Staubli VAL3: BackHomePage.pgx

public program BackHomePage(joint x_jHome, tool x_tTool, mdesc x_mHome)
  local num l_nKey
  local string l_sButton[2]
  local num l_i
  local bool l_bHomeDone
  local bool l_bExit
  local string l_sYesNo
begin
  //-----------------------------------------------------------------------
  //Header begin
  //Description of program
  //  手臂回零页面
  //  F1:终止回零
  //Input parameters
  //
  //Output paramaters
  //Example
  //  call BackHomePage()
  //History
  //  Creation : 2012-06-11 - PF.Zhong
  //Header end
  //-----------------------------------------------------------------------
  cls()
  bHomeDone=false
  l_bExit=false
  taskCreate "BackHome",30,BackHome(x_jHome,x_tTool,x_mHome,bHomeDone)
  delay(0.004)
  while !bHomeDone and !l_bExit
      call user:timerDialog("机器人正回Home点，按住Move/Hold键",0)
      call user:typeLen(1,13,"终止",4)
      l_nKey=getKey()
      switch l_nKey
        case 271
          //终止
          l_sButton[0]="是"
          l_sButton[1]="否"
          call user:questionDialog("是否终止回零?",l_sButton,l_i)
          if l_i==0 or l_i==1
            resetMotion()
            stopMove()
            taskKill("BackHome")
            l_bExit=true
          else
            cls()
            call user:timerDialog("机器人正回Home点，按住Move/Hold键",0)
          endIf
        break
      endSwitch
      delay(0)
    endWhile
  if bHomeDone
    l_sYesNo="确定"
    call user:yes("手臂回零完成!",l_sYesNo)
  else
    l_sYesNo="确定"
    call user:yes("手臂回零未完成!",l_sYesNo)
  endIf
end
